ABB RobotStudio station: huevo_20221021-155345.rsstn

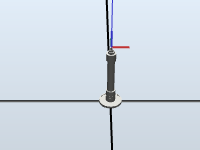
Station Station (saved by RobotStudio 6.5.7558.2005)
Layout (positions relative to the parent item):
  - TOOLSJ [mechanism, from Libraries\HCV2.rslib] at (0, 0, 0) mm
